(* IEC 61131-3 sources: plc_generation_empirical_study/datasets/packages/internal_v0_1/qualification_only/C04_H01_qualified_event_counter, 1 file *)

(* ---- reference.st ---- *)
FUNCTION_BLOCK C04_H01_qualified_event_counter
VAR_INPUT
    Event : BOOL;
    Qualify : BOOL;
    Reset : BOOL;
    MaxCount : INT;
END_VAR
VAR_OUTPUT
    Count : INT;
    AcceptedPulse : BOOL;
    AtLimit : BOOL;
END_VAR
VAR
    PrevEvent : BOOL := FALSE;
END_VAR

AcceptedPulse := FALSE;
IF Reset THEN
    Count := 0;
ELSIF Event AND (NOT PrevEvent) AND Qualify AND (Count < MaxCount) THEN
    Count := Count + 1;
    AcceptedPulse := TRUE;
END_IF;
AtLimit := Count >= MaxCount;
PrevEvent := Event;

END_FUNCTION_BLOCK
